REGION Network 63: BRAKE TEST FAULT AXIS 12
   RUNG wire#powerrail
      Contact( "DB1046_C22_BRAKE_TEST".BRAKE_TEST_ERROR )
      wire#w1
      Contact( #BRAKE_TEST_AXIS_C22 )
      wire#w2
      Coil( "DB1030_TEST_STOP".TEST_STP_TST_BRK_F_AX_12 )
   END_RUNG
   RUNG wire#powerrail
      Contact( "DB1030_TEST_STOP".TEST_STP_SQ_TIME_EXCEEDED )
      Contact( "DB1030_TEST_STOP".TEST_STP_TST_BRK_AX_12 )
   END_RUNG wire#w1
   RUNG wire#powerrail
      Contact( "DB1030_TEST_STOP".TEST_STP_TST_BRK_F_AX_12 )
      I_Contact( "DB2120_MPP_ITC_IPC".RESET_FAULTS )
   END_RUNG wire#w1
   RUNG wire#w2
      Coil( "DB426_ALARMS_WARNINGS".ALARMS.GENERAL."700603" )
   END_RUNG
   // the same network as SCL:
   "DB1030_TEST_STOP".TEST_STP_TST_BRK_F_AX_12 := ("DB1046_C22_BRAKE_TEST".BRAKE_TEST_ERROR OR ("DB1030_TEST_STOP".TEST_STP_SQ_TIME_EXCEEDED AND "DB1030_TEST_STOP".TEST_STP_TST_BRK_AX_12) OR ("DB1030_TEST_STOP".TEST_STP_TST_BRK_F_AX_12 AND NOT "DB2120_MPP_ITC_IPC".RESET_FAULTS)) AND #BRAKE_TEST_AXIS_C22;
   "DB426_ALARMS_WARNINGS".ALARMS.GENERAL."700603" := "DB1030_TEST_STOP".TEST_STP_TST_BRK_F_AX_12;
END_REGION

REGION Network 64: BRAKE TEST FAULT AXIS 13
   RUNG wire#powerrail
      Contact( "DB1047_C23_BRAKE_TEST".BRAKE_TEST_ERROR )
      wire#w1
      Contact( #BRAKE_TEST_AXIS_C23 )
      wire#w2
      Coil( "DB1030_TEST_STOP".TEST_STP_TST_BRK_F_AX_13 )
   END_RUNG
   RUNG wire#powerrail
      Contact( "DB1030_TEST_STOP".TEST_STP_SQ_TIME_EXCEEDED )
      Contact( "DB1030_TEST_STOP".TEST_STP_TST_BRK_AX_13 )
   END_RUNG wire#w1
   RUNG wire#powerrail
      Contact( "DB1030_TEST_STOP".TEST_STP_TST_BRK_F_AX_13 )
      I_Contact( "DB2120_MPP_ITC_IPC".RESET_FAULTS )
   END_RUNG wire#w1
   RUNG wire#w2
      Coil( "DB426_ALARMS_WARNINGS".ALARMS.GENERAL."700604" )
   END_RUNG
   // the same network as SCL:
   "DB1030_TEST_STOP".TEST_STP_TST_BRK_F_AX_13 := ("DB1047_C23_BRAKE_TEST".BRAKE_TEST_ERROR OR ("DB1030_TEST_STOP".TEST_STP_SQ_TIME_EXCEEDED AND "DB1030_TEST_STOP".TEST_STP_TST_BRK_AX_13) OR ("DB1030_TEST_STOP".TEST_STP_TST_BRK_F_AX_13 AND NOT "DB2120_MPP_ITC_IPC".RESET_FAULTS)) AND #BRAKE_TEST_AXIS_C23;
   "DB426_ALARMS_WARNINGS".ALARMS.GENERAL."700604" := "DB1030_TEST_STOP".TEST_STP_TST_BRK_F_AX_13;
END_REGION

REGION Network 65: BRAKE TEST FAULT AXIS 14
   RUNG wire#powerrail
      Contact( "DB1048_C24_BRAKE_TEST".BRAKE_TEST_ERROR )
      wire#w1
      Contact( #BRAKE_TEST_AXIS_C24 )
      wire#w2
      Coil( "DB1030_TEST_STOP".TEST_STP_TST_BRK_F_AX_14 )
   END_RUNG
   RUNG wire#powerrail
      Contact( "DB1030_TEST_STOP".TEST_STP_SQ_TIME_EXCEEDED )
      Contact( "DB1030_TEST_STOP".TEST_STP_TST_BRK_AX_14 )
   END_RUNG wire#w1
   RUNG wire#powerrail
      Contact( "DB1030_TEST_STOP".TEST_STP_TST_BRK_F_AX_14 )
      I_Contact( "DB2120_MPP_ITC_IPC".RESET_FAULTS )
   END_RUNG wire#w1
   RUNG wire#w2
      Coil( "DB426_ALARMS_WARNINGS".ALARMS.GENERAL."700605" )
   END_RUNG
   // the same network as SCL:
   "DB1030_TEST_STOP".TEST_STP_TST_BRK_F_AX_14 := ("DB1048_C24_BRAKE_TEST".BRAKE_TEST_ERROR OR ("DB1030_TEST_STOP".TEST_STP_SQ_TIME_EXCEEDED AND "DB1030_TEST_STOP".TEST_STP_TST_BRK_AX_14) OR ("DB1030_TEST_STOP".TEST_STP_TST_BRK_F_AX_14 AND NOT "DB2120_MPP_ITC_IPC".RESET_FAULTS)) AND #BRAKE_TEST_AXIS_C24;
   "DB426_ALARMS_WARNINGS".ALARMS.GENERAL."700605" := "DB1030_TEST_STOP".TEST_STP_TST_BRK_F_AX_14;
END_REGION

REGION Network 66: BRAKE TEST FAULT AXIS 15
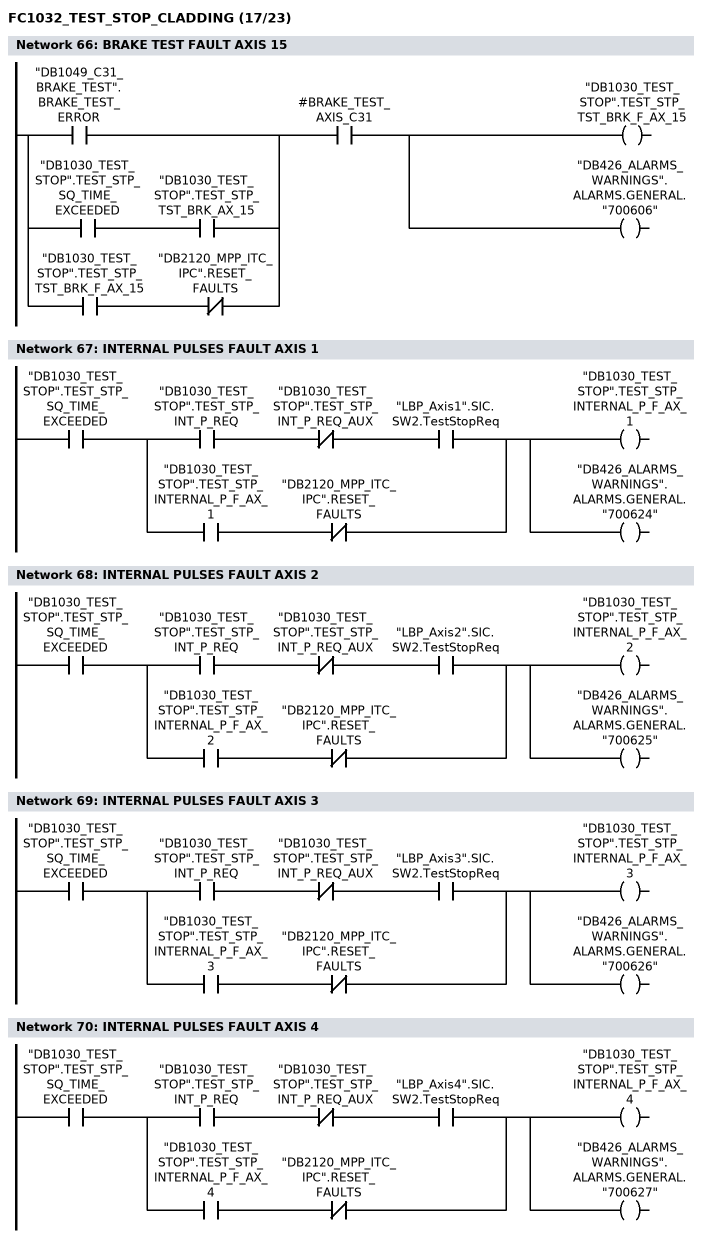
   RUNG wire#powerrail
      Contact( "DB1049_C31_BRAKE_TEST".BRAKE_TEST_ERROR )
      wire#w1
      Contact( #BRAKE_TEST_AXIS_C31 )
      wire#w2
      Coil( "DB1030_TEST_STOP".TEST_STP_TST_BRK_F_AX_15 )
   END_RUNG
   RUNG wire#powerrail
      Contact( "DB1030_TEST_STOP".TEST_STP_SQ_TIME_EXCEEDED )
      Contact( "DB1030_TEST_STOP".TEST_STP_TST_BRK_AX_15 )
   END_RUNG wire#w1
   RUNG wire#powerrail
      Contact( "DB1030_TEST_STOP".TEST_STP_TST_BRK_F_AX_15 )
      I_Contact( "DB2120_MPP_ITC_IPC".RESET_FAULTS )
   END_RUNG wire#w1
   RUNG wire#w2
      Coil( "DB426_ALARMS_WARNINGS".ALARMS.GENERAL."700606" )
   END_RUNG
   // the same network as SCL:
   "DB1030_TEST_STOP".TEST_STP_TST_BRK_F_AX_15 := ("DB1049_C31_BRAKE_TEST".BRAKE_TEST_ERROR OR ("DB1030_TEST_STOP".TEST_STP_SQ_TIME_EXCEEDED AND "DB1030_TEST_STOP".TEST_STP_TST_BRK_AX_15) OR ("DB1030_TEST_STOP".TEST_STP_TST_BRK_F_AX_15 AND NOT "DB2120_MPP_ITC_IPC".RESET_FAULTS)) AND #BRAKE_TEST_AXIS_C31;
   "DB426_ALARMS_WARNINGS".ALARMS.GENERAL."700606" := "DB1030_TEST_STOP".TEST_STP_TST_BRK_F_AX_15;
END_REGION

REGION Network 67: INTERNAL PULSES FAULT AXIS 1
   RUNG wire#powerrail
      Contact( "DB1030_TEST_STOP".TEST_STP_SQ_TIME_EXCEEDED )
      wire#w1
      Contact( "DB1030_TEST_STOP".TEST_STP_INT_P_REQ )
      I_Contact( "DB1030_TEST_STOP".TEST_STP_INT_P_REQ_AUX )
      Contact( "LBP_Axis1".SIC.SW2.TestStopReq )
      wire#w2
      Coil( "DB1030_TEST_STOP".TEST_STP_INTERNAL_P_F_AX_1 )
   END_RUNG
   RUNG wire#w1
      Contact( "DB1030_TEST_STOP".TEST_STP_INTERNAL_P_F_AX_1 )
      I_Contact( "DB2120_MPP_ITC_IPC".RESET_FAULTS )
   END_RUNG wire#w2
   RUNG wire#w2
      Coil( "DB426_ALARMS_WARNINGS".ALARMS.GENERAL."700624" )
   END_RUNG
   // the same network as SCL:
   "DB1030_TEST_STOP".TEST_STP_INTERNAL_P_F_AX_1 := "DB1030_TEST_STOP".TEST_STP_SQ_TIME_EXCEEDED AND (("DB1030_TEST_STOP".TEST_STP_INT_P_REQ AND NOT "DB1030_TEST_STOP".TEST_STP_INT_P_REQ_AUX AND "LBP_Axis1".SIC.SW2.TestStopReq) OR ("DB1030_TEST_STOP".TEST_STP_INTERNAL_P_F_AX_1 AND NOT "DB2120_MPP_ITC_IPC".RESET_FAULTS));
   "DB426_ALARMS_WARNINGS".ALARMS.GENERAL."700624" := "DB1030_TEST_STOP".TEST_STP_INTERNAL_P_F_AX_1;
END_REGION

REGION Network 68: INTERNAL PULSES FAULT AXIS 2
   RUNG wire#powerrail
      Contact( "DB1030_TEST_STOP".TEST_STP_SQ_TIME_EXCEEDED )
      wire#w1
      Contact( "DB1030_TEST_STOP".TEST_STP_INT_P_REQ )
      I_Contact( "DB1030_TEST_STOP".TEST_STP_INT_P_REQ_AUX )
      Contact( "LBP_Axis2".SIC.SW2.TestStopReq )
      wire#w2
      Coil( "DB1030_TEST_STOP".TEST_STP_INTERNAL_P_F_AX_2 )
   END_RUNG
   RUNG wire#w1
      Contact( "DB1030_TEST_STOP".TEST_STP_INTERNAL_P_F_AX_2 )
      I_Contact( "DB2120_MPP_ITC_IPC".RESET_FAULTS )
   END_RUNG wire#w2
   RUNG wire#w2
      Coil( "DB426_ALARMS_WARNINGS".ALARMS.GENERAL."700625" )
   END_RUNG
   // the same network as SCL:
   "DB1030_TEST_STOP".TEST_STP_INTERNAL_P_F_AX_2 := "DB1030_TEST_STOP".TEST_STP_SQ_TIME_EXCEEDED AND (("DB1030_TEST_STOP".TEST_STP_INT_P_REQ AND NOT "DB1030_TEST_STOP".TEST_STP_INT_P_REQ_AUX AND "LBP_Axis2".SIC.SW2.TestStopReq) OR ("DB1030_TEST_STOP".TEST_STP_INTERNAL_P_F_AX_2 AND NOT "DB2120_MPP_ITC_IPC".RESET_FAULTS));
   "DB426_ALARMS_WARNINGS".ALARMS.GENERAL."700625" := "DB1030_TEST_STOP".TEST_STP_INTERNAL_P_F_AX_2;
END_REGION

REGION Network 69: INTERNAL PULSES FAULT AXIS 3
   RUNG wire#powerrail
      Contact( "DB1030_TEST_STOP".TEST_STP_SQ_TIME_EXCEEDED )
      wire#w1
      Contact( "DB1030_TEST_STOP".TEST_STP_INT_P_REQ )
      I_Contact( "DB1030_TEST_STOP".TEST_STP_INT_P_REQ_AUX )
      Contact( "LBP_Axis3".SIC.SW2.TestStopReq )
      wire#w2
      Coil( "DB1030_TEST_STOP".TEST_STP_INTERNAL_P_F_AX_3 )
   END_RUNG
   RUNG wire#w1
      Contact( "DB1030_TEST_STOP".TEST_STP_INTERNAL_P_F_AX_3 )
      I_Contact( "DB2120_MPP_ITC_IPC".RESET_FAULTS )
   END_RUNG wire#w2
   RUNG wire#w2
      Coil( "DB426_ALARMS_WARNINGS".ALARMS.GENERAL."700626" )
   END_RUNG
   // the same network as SCL:
   "DB1030_TEST_STOP".TEST_STP_INTERNAL_P_F_AX_3 := "DB1030_TEST_STOP".TEST_STP_SQ_TIME_EXCEEDED AND (("DB1030_TEST_STOP".TEST_STP_INT_P_REQ AND NOT "DB1030_TEST_STOP".TEST_STP_INT_P_REQ_AUX AND "LBP_Axis3".SIC.SW2.TestStopReq) OR ("DB1030_TEST_STOP".TEST_STP_INTERNAL_P_F_AX_3 AND NOT "DB2120_MPP_ITC_IPC".RESET_FAULTS));
   "DB426_ALARMS_WARNINGS".ALARMS.GENERAL."700626" := "DB1030_TEST_STOP".TEST_STP_INTERNAL_P_F_AX_3;
END_REGION

REGION Network 70: INTERNAL PULSES FAULT AXIS 4
   RUNG wire#powerrail
      Contact( "DB1030_TEST_STOP".TEST_STP_SQ_TIME_EXCEEDED )
      wire#w1
      Contact( "DB1030_TEST_STOP".TEST_STP_INT_P_REQ )
      I_Contact( "DB1030_TEST_STOP".TEST_STP_INT_P_REQ_AUX )
      Contact( "LBP_Axis4".SIC.SW2.TestStopReq )
      wire#w2
      Coil( "DB1030_TEST_STOP".TEST_STP_INTERNAL_P_F_AX_4 )
   END_RUNG
   RUNG wire#w1
      Contact( "DB1030_TEST_STOP".TEST_STP_INTERNAL_P_F_AX_4 )
      I_Contact( "DB2120_MPP_ITC_IPC".RESET_FAULTS )
   END_RUNG wire#w2
   RUNG wire#w2
      Coil( "DB426_ALARMS_WARNINGS".ALARMS.GENERAL."700627" )
   END_RUNG
   // the same network as SCL:
   "DB1030_TEST_STOP".TEST_STP_INTERNAL_P_F_AX_4 := "DB1030_TEST_STOP".TEST_STP_SQ_TIME_EXCEEDED AND (("DB1030_TEST_STOP".TEST_STP_INT_P_REQ AND NOT "DB1030_TEST_STOP".TEST_STP_INT_P_REQ_AUX AND "LBP_Axis4".SIC.SW2.TestStopReq) OR ("DB1030_TEST_STOP".TEST_STP_INTERNAL_P_F_AX_4 AND NOT "DB2120_MPP_ITC_IPC".RESET_FAULTS));
   "DB426_ALARMS_WARNINGS".ALARMS.GENERAL."700627" := "DB1030_TEST_STOP".TEST_STP_INTERNAL_P_F_AX_4;
END_REGION

REGION Network 71: INTERNAL PULSES FAULT AXIS 5
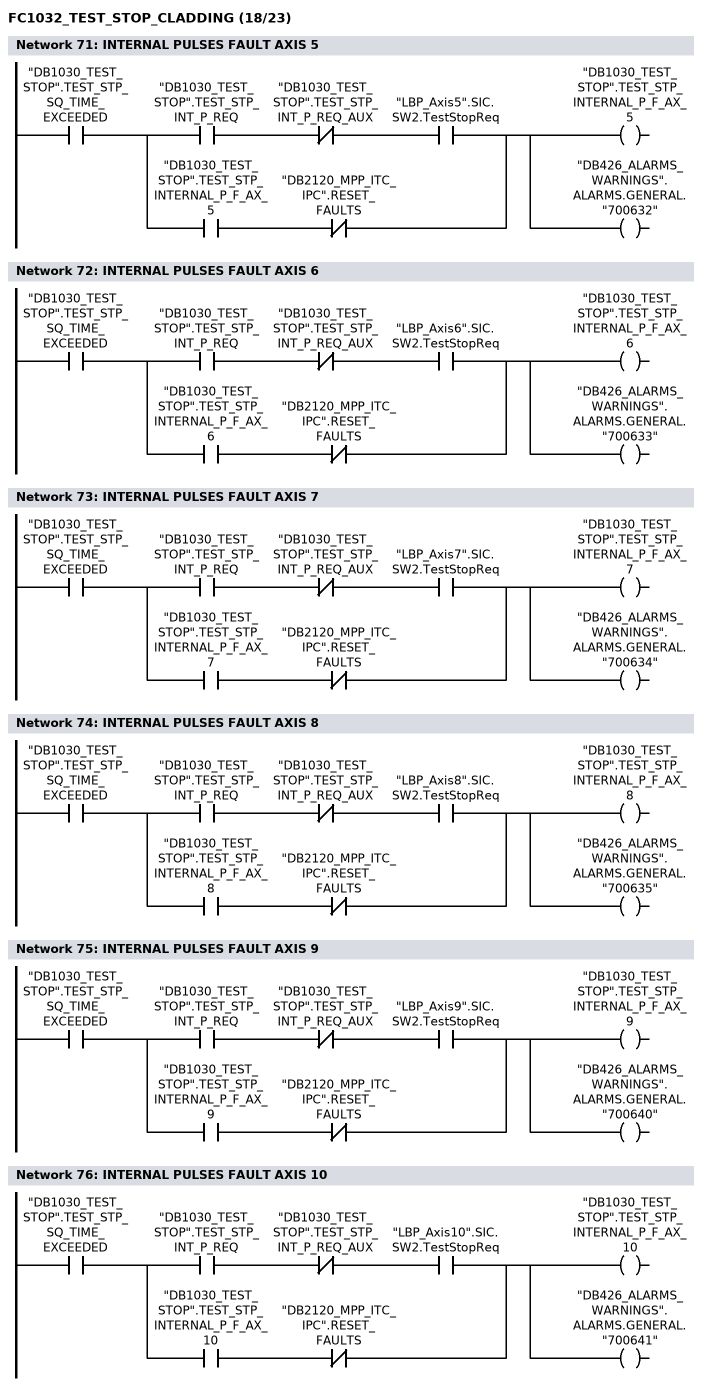
   RUNG wire#powerrail
      Contact( "DB1030_TEST_STOP".TEST_STP_SQ_TIME_EXCEEDED )
      wire#w1
      Contact( "DB1030_TEST_STOP".TEST_STP_INT_P_REQ )
      I_Contact( "DB1030_TEST_STOP".TEST_STP_INT_P_REQ_AUX )
      Contact( "LBP_Axis5".SIC.SW2.TestStopReq )
      wire#w2
      Coil( "DB1030_TEST_STOP".TEST_STP_INTERNAL_P_F_AX_5 )
   END_RUNG
   RUNG wire#w1
      Contact( "DB1030_TEST_STOP".TEST_STP_INTERNAL_P_F_AX_5 )
      I_Contact( "DB2120_MPP_ITC_IPC".RESET_FAULTS )
   END_RUNG wire#w2
   RUNG wire#w2
      Coil( "DB426_ALARMS_WARNINGS".ALARMS.GENERAL."700632" )
   END_RUNG
   // the same network as SCL:
   "DB1030_TEST_STOP".TEST_STP_INTERNAL_P_F_AX_5 := "DB1030_TEST_STOP".TEST_STP_SQ_TIME_EXCEEDED AND (("DB1030_TEST_STOP".TEST_STP_INT_P_REQ AND NOT "DB1030_TEST_STOP".TEST_STP_INT_P_REQ_AUX AND "LBP_Axis5".SIC.SW2.TestStopReq) OR ("DB1030_TEST_STOP".TEST_STP_INTERNAL_P_F_AX_5 AND NOT "DB2120_MPP_ITC_IPC".RESET_FAULTS));
   "DB426_ALARMS_WARNINGS".ALARMS.GENERAL."700632" := "DB1030_TEST_STOP".TEST_STP_INTERNAL_P_F_AX_5;
END_REGION

REGION Network 72: INTERNAL PULSES FAULT AXIS 6
   RUNG wire#powerrail
      Contact( "DB1030_TEST_STOP".TEST_STP_SQ_TIME_EXCEEDED )
      wire#w1
      Contact( "DB1030_TEST_STOP".TEST_STP_INT_P_REQ )
      I_Contact( "DB1030_TEST_STOP".TEST_STP_INT_P_REQ_AUX )
      Contact( "LBP_Axis6".SIC.SW2.TestStopReq )
      wire#w2
      Coil( "DB1030_TEST_STOP".TEST_STP_INTERNAL_P_F_AX_6 )
   END_RUNG
   RUNG wire#w1
      Contact( "DB1030_TEST_STOP".TEST_STP_INTERNAL_P_F_AX_6 )
      I_Contact( "DB2120_MPP_ITC_IPC".RESET_FAULTS )
   END_RUNG wire#w2
   RUNG wire#w2
      Coil( "DB426_ALARMS_WARNINGS".ALARMS.GENERAL."700633" )
   END_RUNG
   // the same network as SCL:
   "DB1030_TEST_STOP".TEST_STP_INTERNAL_P_F_AX_6 := "DB1030_TEST_STOP".TEST_STP_SQ_TIME_EXCEEDED AND (("DB1030_TEST_STOP".TEST_STP_INT_P_REQ AND NOT "DB1030_TEST_STOP".TEST_STP_INT_P_REQ_AUX AND "LBP_Axis6".SIC.SW2.TestStopReq) OR ("DB1030_TEST_STOP".TEST_STP_INTERNAL_P_F_AX_6 AND NOT "DB2120_MPP_ITC_IPC".RESET_FAULTS));
   "DB426_ALARMS_WARNINGS".ALARMS.GENERAL."700633" := "DB1030_TEST_STOP".TEST_STP_INTERNAL_P_F_AX_6;
END_REGION

REGION Network 73: INTERNAL PULSES FAULT AXIS 7
   RUNG wire#powerrail
      Contact( "DB1030_TEST_STOP".TEST_STP_SQ_TIME_EXCEEDED )
      wire#w1
      Contact( "DB1030_TEST_STOP".TEST_STP_INT_P_REQ )
      I_Contact( "DB1030_TEST_STOP".TEST_STP_INT_P_REQ_AUX )
      Contact( "LBP_Axis7".SIC.SW2.TestStopReq )
      wire#w2
      Coil( "DB1030_TEST_STOP".TEST_STP_INTERNAL_P_F_AX_7 )
   END_RUNG
   RUNG wire#w1
      Contact( "DB1030_TEST_STOP".TEST_STP_INTERNAL_P_F_AX_7 )
      I_Contact( "DB2120_MPP_ITC_IPC".RESET_FAULTS )
   END_RUNG wire#w2
   RUNG wire#w2
      Coil( "DB426_ALARMS_WARNINGS".ALARMS.GENERAL."700634" )
   END_RUNG
   // the same network as SCL:
   "DB1030_TEST_STOP".TEST_STP_INTERNAL_P_F_AX_7 := "DB1030_TEST_STOP".TEST_STP_SQ_TIME_EXCEEDED AND (("DB1030_TEST_STOP".TEST_STP_INT_P_REQ AND NOT "DB1030_TEST_STOP".TEST_STP_INT_P_REQ_AUX AND "LBP_Axis7".SIC.SW2.TestStopReq) OR ("DB1030_TEST_STOP".TEST_STP_INTERNAL_P_F_AX_7 AND NOT "DB2120_MPP_ITC_IPC".RESET_FAULTS));
   "DB426_ALARMS_WARNINGS".ALARMS.GENERAL."700634" := "DB1030_TEST_STOP".TEST_STP_INTERNAL_P_F_AX_7;
END_REGION

REGION Network 74: INTERNAL PULSES FAULT AXIS 8
   RUNG wire#powerrail
      Contact( "DB1030_TEST_STOP".TEST_STP_SQ_TIME_EXCEEDED )
      wire#w1
      Contact( "DB1030_TEST_STOP".TEST_STP_INT_P_REQ )
      I_Contact( "DB1030_TEST_STOP".TEST_STP_INT_P_REQ_AUX )
      Contact( "LBP_Axis8".SIC.SW2.TestStopReq )
      wire#w2
      Coil( "DB1030_TEST_STOP".TEST_STP_INTERNAL_P_F_AX_8 )
   END_RUNG
   RUNG wire#w1
      Contact( "DB1030_TEST_STOP".TEST_STP_INTERNAL_P_F_AX_8 )
      I_Contact( "DB2120_MPP_ITC_IPC".RESET_FAULTS )
   END_RUNG wire#w2
   RUNG wire#w2
      Coil( "DB426_ALARMS_WARNINGS".ALARMS.GENERAL."700635" )
   END_RUNG
   // the same network as SCL:
   "DB1030_TEST_STOP".TEST_STP_INTERNAL_P_F_AX_8 := "DB1030_TEST_STOP".TEST_STP_SQ_TIME_EXCEEDED AND (("DB1030_TEST_STOP".TEST_STP_INT_P_REQ AND NOT "DB1030_TEST_STOP".TEST_STP_INT_P_REQ_AUX AND "LBP_Axis8".SIC.SW2.TestStopReq) OR ("DB1030_TEST_STOP".TEST_STP_INTERNAL_P_F_AX_8 AND NOT "DB2120_MPP_ITC_IPC".RESET_FAULTS));
   "DB426_ALARMS_WARNINGS".ALARMS.GENERAL."700635" := "DB1030_TEST_STOP".TEST_STP_INTERNAL_P_F_AX_8;
END_REGION

REGION Network 75: INTERNAL PULSES FAULT AXIS 9
   RUNG wire#powerrail
      Contact( "DB1030_TEST_STOP".TEST_STP_SQ_TIME_EXCEEDED )
      wire#w1
      Contact( "DB1030_TEST_STOP".TEST_STP_INT_P_REQ )
      I_Contact( "DB1030_TEST_STOP".TEST_STP_INT_P_REQ_AUX )
      Contact( "LBP_Axis9".SIC.SW2.TestStopReq )
      wire#w2
      Coil( "DB1030_TEST_STOP".TEST_STP_INTERNAL_P_F_AX_9 )
   END_RUNG
   RUNG wire#w1
      Contact( "DB1030_TEST_STOP".TEST_STP_INTERNAL_P_F_AX_9 )
      I_Contact( "DB2120_MPP_ITC_IPC".RESET_FAULTS )
   END_RUNG wire#w2
   RUNG wire#w2
      Coil( "DB426_ALARMS_WARNINGS".ALARMS.GENERAL."700640" )
   END_RUNG
   // the same network as SCL:
   "DB1030_TEST_STOP".TEST_STP_INTERNAL_P_F_AX_9 := "DB1030_TEST_STOP".TEST_STP_SQ_TIME_EXCEEDED AND (("DB1030_TEST_STOP".TEST_STP_INT_P_REQ AND NOT "DB1030_TEST_STOP".TEST_STP_INT_P_REQ_AUX AND "LBP_Axis9".SIC.SW2.TestStopReq) OR ("DB1030_TEST_STOP".TEST_STP_INTERNAL_P_F_AX_9 AND NOT "DB2120_MPP_ITC_IPC".RESET_FAULTS));
   "DB426_ALARMS_WARNINGS".ALARMS.GENERAL."700640" := "DB1030_TEST_STOP".TEST_STP_INTERNAL_P_F_AX_9;
END_REGION

REGION Network 76: INTERNAL PULSES FAULT AXIS 10
   RUNG wire#powerrail
      Contact( "DB1030_TEST_STOP".TEST_STP_SQ_TIME_EXCEEDED )
      wire#w1
      Contact( "DB1030_TEST_STOP".TEST_STP_INT_P_REQ )
      I_Contact( "DB1030_TEST_STOP".TEST_STP_INT_P_REQ_AUX )
      Contact( "LBP_Axis10".SIC.SW2.TestStopReq )
      wire#w2
      Coil( "DB1030_TEST_STOP".TEST_STP_INTERNAL_P_F_AX_10 )
   END_RUNG
   RUNG wire#w1
      Contact( "DB1030_TEST_STOP".TEST_STP_INTERNAL_P_F_AX_10 )
      I_Contact( "DB2120_MPP_ITC_IPC".RESET_FAULTS )
   END_RUNG wire#w2
   RUNG wire#w2
      Coil( "DB426_ALARMS_WARNINGS".ALARMS.GENERAL."700641" )
   END_RUNG
   // the same network as SCL:
   "DB1030_TEST_STOP".TEST_STP_INTERNAL_P_F_AX_10 := "DB1030_TEST_STOP".TEST_STP_SQ_TIME_EXCEEDED AND (("DB1030_TEST_STOP".TEST_STP_INT_P_REQ AND NOT "DB1030_TEST_STOP".TEST_STP_INT_P_REQ_AUX AND "LBP_Axis10".SIC.SW2.TestStopReq) OR ("DB1030_TEST_STOP".TEST_STP_INTERNAL_P_F_AX_10 AND NOT "DB2120_MPP_ITC_IPC".RESET_FAULTS));
   "DB426_ALARMS_WARNINGS".ALARMS.GENERAL."700641" := "DB1030_TEST_STOP".TEST_STP_INTERNAL_P_F_AX_10;
END_REGION

REGION Network 77: INTERNAL PULSES FAULT AXIS 11
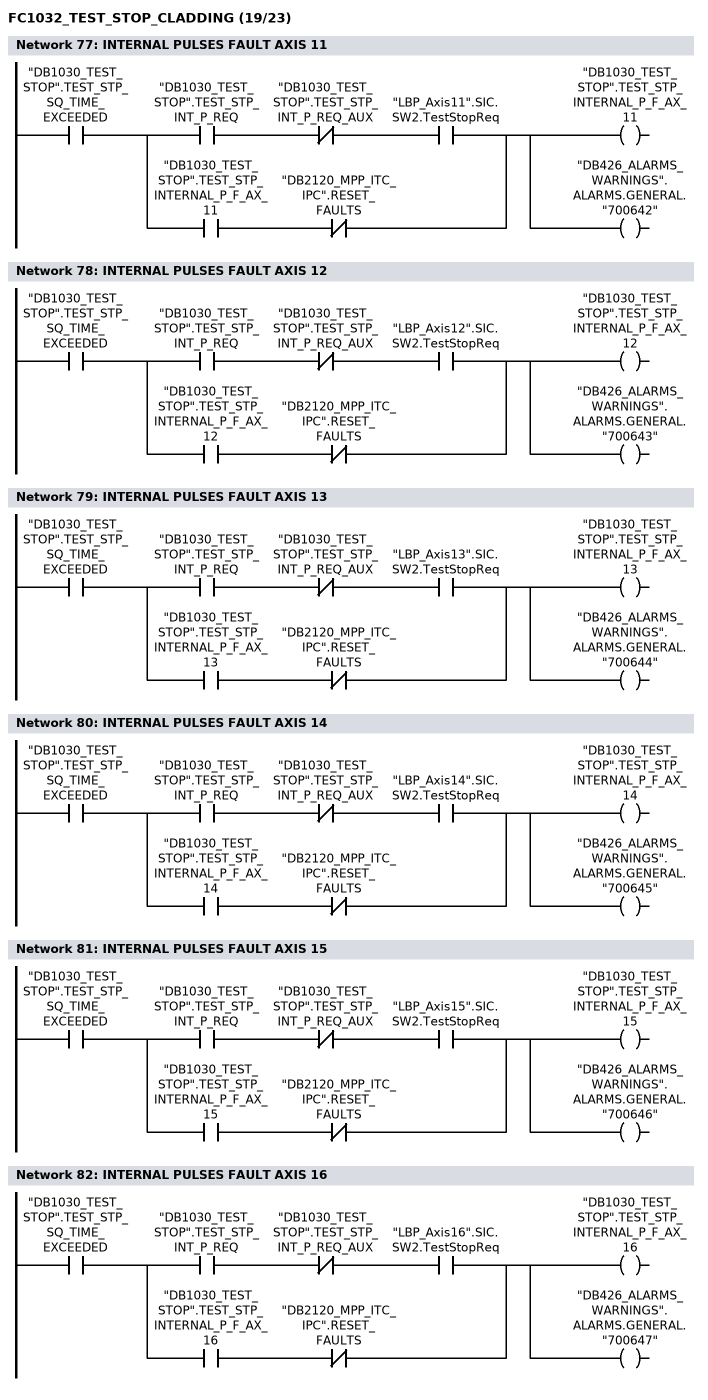
   RUNG wire#powerrail
      Contact( "DB1030_TEST_STOP".TEST_STP_SQ_TIME_EXCEEDED )
      wire#w1
      Contact( "DB1030_TEST_STOP".TEST_STP_INT_P_REQ )
      I_Contact( "DB1030_TEST_STOP".TEST_STP_INT_P_REQ_AUX )
      Contact( "LBP_Axis11".SIC.SW2.TestStopReq )
      wire#w2
      Coil( "DB1030_TEST_STOP".TEST_STP_INTERNAL_P_F_AX_11 )
   END_RUNG
   RUNG wire#w1
      Contact( "DB1030_TEST_STOP".TEST_STP_INTERNAL_P_F_AX_11 )
      I_Contact( "DB2120_MPP_ITC_IPC".RESET_FAULTS )
   END_RUNG wire#w2
   RUNG wire#w2
      Coil( "DB426_ALARMS_WARNINGS".ALARMS.GENERAL."700642" )
   END_RUNG
   // the same network as SCL:
   "DB1030_TEST_STOP".TEST_STP_INTERNAL_P_F_AX_11 := "DB1030_TEST_STOP".TEST_STP_SQ_TIME_EXCEEDED AND (("DB1030_TEST_STOP".TEST_STP_INT_P_REQ AND NOT "DB1030_TEST_STOP".TEST_STP_INT_P_REQ_AUX AND "LBP_Axis11".SIC.SW2.TestStopReq) OR ("DB1030_TEST_STOP".TEST_STP_INTERNAL_P_F_AX_11 AND NOT "DB2120_MPP_ITC_IPC".RESET_FAULTS));
   "DB426_ALARMS_WARNINGS".ALARMS.GENERAL."700642" := "DB1030_TEST_STOP".TEST_STP_INTERNAL_P_F_AX_11;
END_REGION

REGION Network 78: INTERNAL PULSES FAULT AXIS 12
   RUNG wire#powerrail
      Contact( "DB1030_TEST_STOP".TEST_STP_SQ_TIME_EXCEEDED )
      wire#w1
      Contact( "DB1030_TEST_STOP".TEST_STP_INT_P_REQ )
      I_Contact( "DB1030_TEST_STOP".TEST_STP_INT_P_REQ_AUX )
      Contact( "LBP_Axis12".SIC.SW2.TestStopReq )
      wire#w2
      Coil( "DB1030_TEST_STOP".TEST_STP_INTERNAL_P_F_AX_12 )
   END_RUNG
   RUNG wire#w1
      Contact( "DB1030_TEST_STOP".TEST_STP_INTERNAL_P_F_AX_12 )
      I_Contact( "DB2120_MPP_ITC_IPC".RESET_FAULTS )
   END_RUNG wire#w2
   RUNG wire#w2
      Coil( "DB426_ALARMS_WARNINGS".ALARMS.GENERAL."700643" )
   END_RUNG
   // the same network as SCL:
   "DB1030_TEST_STOP".TEST_STP_INTERNAL_P_F_AX_12 := "DB1030_TEST_STOP".TEST_STP_SQ_TIME_EXCEEDED AND (("DB1030_TEST_STOP".TEST_STP_INT_P_REQ AND NOT "DB1030_TEST_STOP".TEST_STP_INT_P_REQ_AUX AND "LBP_Axis12".SIC.SW2.TestStopReq) OR ("DB1030_TEST_STOP".TEST_STP_INTERNAL_P_F_AX_12 AND NOT "DB2120_MPP_ITC_IPC".RESET_FAULTS));
   "DB426_ALARMS_WARNINGS".ALARMS.GENERAL."700643" := "DB1030_TEST_STOP".TEST_STP_INTERNAL_P_F_AX_12;
END_REGION

REGION Network 79: INTERNAL PULSES FAULT AXIS 13
   RUNG wire#powerrail
      Contact( "DB1030_TEST_STOP".TEST_STP_SQ_TIME_EXCEEDED )
      wire#w1
      Contact( "DB1030_TEST_STOP".TEST_STP_INT_P_REQ )
      I_Contact( "DB1030_TEST_STOP".TEST_STP_INT_P_REQ_AUX )
      Contact( "LBP_Axis13".SIC.SW2.TestStopReq )
      wire#w2
      Coil( "DB1030_TEST_STOP".TEST_STP_INTERNAL_P_F_AX_13 )
   END_RUNG
   RUNG wire#w1
      Contact( "DB1030_TEST_STOP".TEST_STP_INTERNAL_P_F_AX_13 )
      I_Contact( "DB2120_MPP_ITC_IPC".RESET_FAULTS )
   END_RUNG wire#w2
   RUNG wire#w2
      Coil( "DB426_ALARMS_WARNINGS".ALARMS.GENERAL."700644" )
   END_RUNG
   // the same network as SCL:
   "DB1030_TEST_STOP".TEST_STP_INTERNAL_P_F_AX_13 := "DB1030_TEST_STOP".TEST_STP_SQ_TIME_EXCEEDED AND (("DB1030_TEST_STOP".TEST_STP_INT_P_REQ AND NOT "DB1030_TEST_STOP".TEST_STP_INT_P_REQ_AUX AND "LBP_Axis13".SIC.SW2.TestStopReq) OR ("DB1030_TEST_STOP".TEST_STP_INTERNAL_P_F_AX_13 AND NOT "DB2120_MPP_ITC_IPC".RESET_FAULTS));
   "DB426_ALARMS_WARNINGS".ALARMS.GENERAL."700644" := "DB1030_TEST_STOP".TEST_STP_INTERNAL_P_F_AX_13;
END_REGION

REGION Network 80: INTERNAL PULSES FAULT AXIS 14
   RUNG wire#powerrail
      Contact( "DB1030_TEST_STOP".TEST_STP_SQ_TIME_EXCEEDED )
      wire#w1
      Contact( "DB1030_TEST_STOP".TEST_STP_INT_P_REQ )
      I_Contact( "DB1030_TEST_STOP".TEST_STP_INT_P_REQ_AUX )
      Contact( "LBP_Axis14".SIC.SW2.TestStopReq )
      wire#w2
      Coil( "DB1030_TEST_STOP".TEST_STP_INTERNAL_P_F_AX_14 )
   END_RUNG
   RUNG wire#w1
      Contact( "DB1030_TEST_STOP".TEST_STP_INTERNAL_P_F_AX_14 )
      I_Contact( "DB2120_MPP_ITC_IPC".RESET_FAULTS )
   END_RUNG wire#w2
   RUNG wire#w2
      Coil( "DB426_ALARMS_WARNINGS".ALARMS.GENERAL."700645" )
   END_RUNG
   // the same network as SCL:
   "DB1030_TEST_STOP".TEST_STP_INTERNAL_P_F_AX_14 := "DB1030_TEST_STOP".TEST_STP_SQ_TIME_EXCEEDED AND (("DB1030_TEST_STOP".TEST_STP_INT_P_REQ AND NOT "DB1030_TEST_STOP".TEST_STP_INT_P_REQ_AUX AND "LBP_Axis14".SIC.SW2.TestStopReq) OR ("DB1030_TEST_STOP".TEST_STP_INTERNAL_P_F_AX_14 AND NOT "DB2120_MPP_ITC_IPC".RESET_FAULTS));
   "DB426_ALARMS_WARNINGS".ALARMS.GENERAL."700645" := "DB1030_TEST_STOP".TEST_STP_INTERNAL_P_F_AX_14;
END_REGION

REGION Network 81: INTERNAL PULSES FAULT AXIS 15
   RUNG wire#powerrail
      Contact( "DB1030_TEST_STOP".TEST_STP_SQ_TIME_EXCEEDED )
      wire#w1
      Contact( "DB1030_TEST_STOP".TEST_STP_INT_P_REQ )
      I_Contact( "DB1030_TEST_STOP".TEST_STP_INT_P_REQ_AUX )
      Contact( "LBP_Axis15".SIC.SW2.TestStopReq )
      wire#w2
      Coil( "DB1030_TEST_STOP".TEST_STP_INTERNAL_P_F_AX_15 )
   END_RUNG
   RUNG wire#w1
      Contact( "DB1030_TEST_STOP".TEST_STP_INTERNAL_P_F_AX_15 )
      I_Contact( "DB2120_MPP_ITC_IPC".RESET_FAULTS )
   END_RUNG wire#w2
   RUNG wire#w2
      Coil( "DB426_ALARMS_WARNINGS".ALARMS.GENERAL."700646" )
   END_RUNG
   // the same network as SCL:
   "DB1030_TEST_STOP".TEST_STP_INTERNAL_P_F_AX_15 := "DB1030_TEST_STOP".TEST_STP_SQ_TIME_EXCEEDED AND (("DB1030_TEST_STOP".TEST_STP_INT_P_REQ AND NOT "DB1030_TEST_STOP".TEST_STP_INT_P_REQ_AUX AND "LBP_Axis15".SIC.SW2.TestStopReq) OR ("DB1030_TEST_STOP".TEST_STP_INTERNAL_P_F_AX_15 AND NOT "DB2120_MPP_ITC_IPC".RESET_FAULTS));
   "DB426_ALARMS_WARNINGS".ALARMS.GENERAL."700646" := "DB1030_TEST_STOP".TEST_STP_INTERNAL_P_F_AX_15;
END_REGION

REGION Network 82: INTERNAL PULSES FAULT AXIS 16
   RUNG wire#powerrail
      Contact( "DB1030_TEST_STOP".TEST_STP_SQ_TIME_EXCEEDED )
      wire#w1
      Contact( "DB1030_TEST_STOP".TEST_STP_INT_P_REQ )
      I_Contact( "DB1030_TEST_STOP".TEST_STP_INT_P_REQ_AUX )
      Contact( "LBP_Axis16".SIC.SW2.TestStopReq )
      wire#w2
      Coil( "DB1030_TEST_STOP".TEST_STP_INTERNAL_P_F_AX_16 )
   END_RUNG
   RUNG wire#w1
      Contact( "DB1030_TEST_STOP".TEST_STP_INTERNAL_P_F_AX_16 )
      I_Contact( "DB2120_MPP_ITC_IPC".RESET_FAULTS )
   END_RUNG wire#w2
   RUNG wire#w2
      Coil( "DB426_ALARMS_WARNINGS".ALARMS.GENERAL."700647" )
   END_RUNG
   // the same network as SCL:
   "DB1030_TEST_STOP".TEST_STP_INTERNAL_P_F_AX_16 := "DB1030_TEST_STOP".TEST_STP_SQ_TIME_EXCEEDED AND (("DB1030_TEST_STOP".TEST_STP_INT_P_REQ AND NOT "DB1030_TEST_STOP".TEST_STP_INT_P_REQ_AUX AND "LBP_Axis16".SIC.SW2.TestStopReq) OR ("DB1030_TEST_STOP".TEST_STP_INTERNAL_P_F_AX_16 AND NOT "DB2120_MPP_ITC_IPC".RESET_FAULTS));
   "DB426_ALARMS_WARNINGS".ALARMS.GENERAL."700647" := "DB1030_TEST_STOP".TEST_STP_INTERNAL_P_F_AX_16;
END_REGION

REGION Network 83: INTERNAL PULSES FAULT AXIS 17
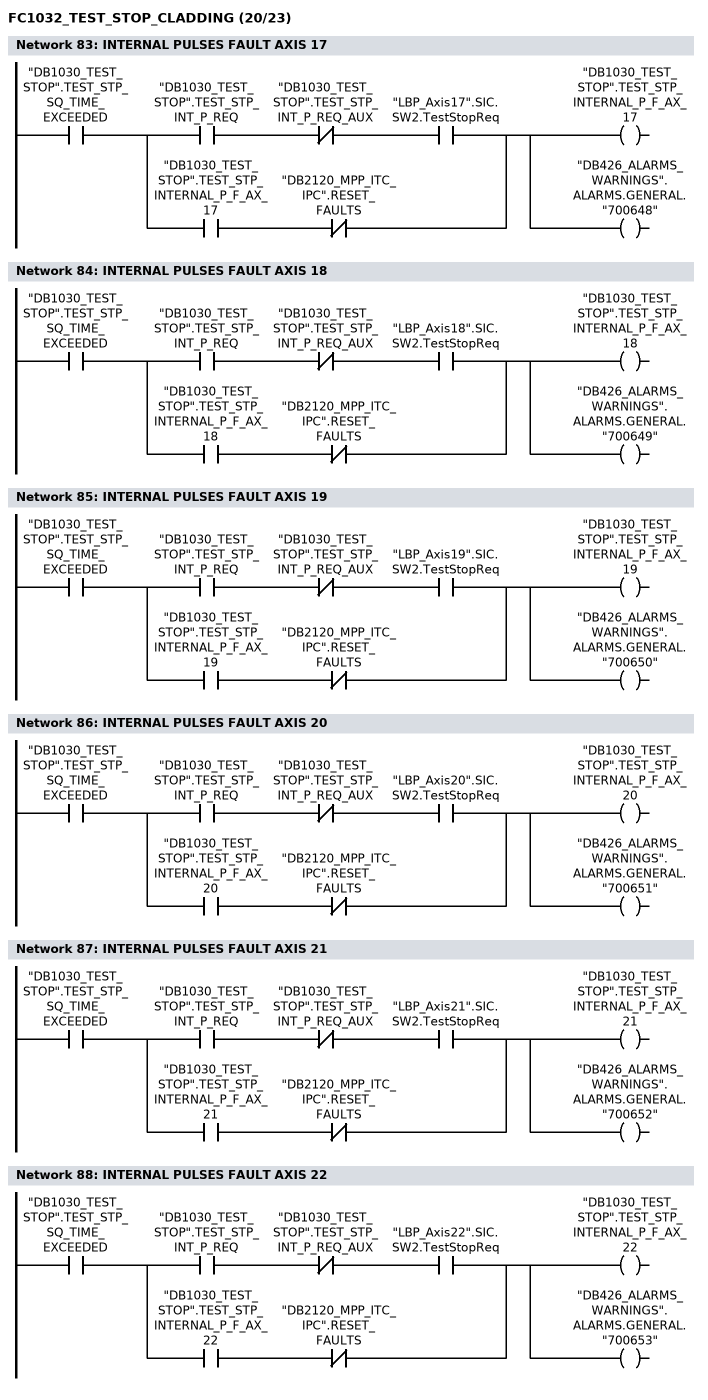
   RUNG wire#powerrail
      Contact( "DB1030_TEST_STOP".TEST_STP_SQ_TIME_EXCEEDED )
      wire#w1
      Contact( "DB1030_TEST_STOP".TEST_STP_INT_P_REQ )
      I_Contact( "DB1030_TEST_STOP".TEST_STP_INT_P_REQ_AUX )
      Contact( "LBP_Axis17".SIC.SW2.TestStopReq )
      wire#w2
      Coil( "DB1030_TEST_STOP".TEST_STP_INTERNAL_P_F_AX_17 )
   END_RUNG
   RUNG wire#w1
      Contact( "DB1030_TEST_STOP".TEST_STP_INTERNAL_P_F_AX_17 )
      I_Contact( "DB2120_MPP_ITC_IPC".RESET_FAULTS )
   END_RUNG wire#w2
   RUNG wire#w2
      Coil( "DB426_ALARMS_WARNINGS".ALARMS.GENERAL."700648" )
   END_RUNG
   // the same network as SCL:
   "DB1030_TEST_STOP".TEST_STP_INTERNAL_P_F_AX_17 := "DB1030_TEST_STOP".TEST_STP_SQ_TIME_EXCEEDED AND (("DB1030_TEST_STOP".TEST_STP_INT_P_REQ AND NOT "DB1030_TEST_STOP".TEST_STP_INT_P_REQ_AUX AND "LBP_Axis17".SIC.SW2.TestStopReq) OR ("DB1030_TEST_STOP".TEST_STP_INTERNAL_P_F_AX_17 AND NOT "DB2120_MPP_ITC_IPC".RESET_FAULTS));
   "DB426_ALARMS_WARNINGS".ALARMS.GENERAL."700648" := "DB1030_TEST_STOP".TEST_STP_INTERNAL_P_F_AX_17;
END_REGION

REGION Network 84: INTERNAL PULSES FAULT AXIS 18
   RUNG wire#powerrail
      Contact( "DB1030_TEST_STOP".TEST_STP_SQ_TIME_EXCEEDED )
      wire#w1
      Contact( "DB1030_TEST_STOP".TEST_STP_INT_P_REQ )
      I_Contact( "DB1030_TEST_STOP".TEST_STP_INT_P_REQ_AUX )
      Contact( "LBP_Axis18".SIC.SW2.TestStopReq )
      wire#w2
      Coil( "DB1030_TEST_STOP".TEST_STP_INTERNAL_P_F_AX_18 )
   END_RUNG
   RUNG wire#w1
      Contact( "DB1030_TEST_STOP".TEST_STP_INTERNAL_P_F_AX_18 )
      I_Contact( "DB2120_MPP_ITC_IPC".RESET_FAULTS )
   END_RUNG wire#w2
   RUNG wire#w2
      Coil( "DB426_ALARMS_WARNINGS".ALARMS.GENERAL."700649" )
   END_RUNG
   // the same network as SCL:
   "DB1030_TEST_STOP".TEST_STP_INTERNAL_P_F_AX_18 := "DB1030_TEST_STOP".TEST_STP_SQ_TIME_EXCEEDED AND (("DB1030_TEST_STOP".TEST_STP_INT_P_REQ AND NOT "DB1030_TEST_STOP".TEST_STP_INT_P_REQ_AUX AND "LBP_Axis18".SIC.SW2.TestStopReq) OR ("DB1030_TEST_STOP".TEST_STP_INTERNAL_P_F_AX_18 AND NOT "DB2120_MPP_ITC_IPC".RESET_FAULTS));
   "DB426_ALARMS_WARNINGS".ALARMS.GENERAL."700649" := "DB1030_TEST_STOP".TEST_STP_INTERNAL_P_F_AX_18;
END_REGION

REGION Network 85: INTERNAL PULSES FAULT AXIS 19
   RUNG wire#powerrail
      Contact( "DB1030_TEST_STOP".TEST_STP_SQ_TIME_EXCEEDED )
      wire#w1
      Contact( "DB1030_TEST_STOP".TEST_STP_INT_P_REQ )
      I_Contact( "DB1030_TEST_STOP".TEST_STP_INT_P_REQ_AUX )
      Contact( "LBP_Axis19".SIC.SW2.TestStopReq )
      wire#w2
      Coil( "DB1030_TEST_STOP".TEST_STP_INTERNAL_P_F_AX_19 )
   END_RUNG
   RUNG wire#w1
      Contact( "DB1030_TEST_STOP".TEST_STP_INTERNAL_P_F_AX_19 )
      I_Contact( "DB2120_MPP_ITC_IPC".RESET_FAULTS )
   END_RUNG wire#w2
   RUNG wire#w2
      Coil( "DB426_ALARMS_WARNINGS".ALARMS.GENERAL."700650" )
   END_RUNG
   // the same network as SCL:
   "DB1030_TEST_STOP".TEST_STP_INTERNAL_P_F_AX_19 := "DB1030_TEST_STOP".TEST_STP_SQ_TIME_EXCEEDED AND (("DB1030_TEST_STOP".TEST_STP_INT_P_REQ AND NOT "DB1030_TEST_STOP".TEST_STP_INT_P_REQ_AUX AND "LBP_Axis19".SIC.SW2.TestStopReq) OR ("DB1030_TEST_STOP".TEST_STP_INTERNAL_P_F_AX_19 AND NOT "DB2120_MPP_ITC_IPC".RESET_FAULTS));
   "DB426_ALARMS_WARNINGS".ALARMS.GENERAL."700650" := "DB1030_TEST_STOP".TEST_STP_INTERNAL_P_F_AX_19;
END_REGION

REGION Network 86: INTERNAL PULSES FAULT AXIS 20
   RUNG wire#powerrail
      Contact( "DB1030_TEST_STOP".TEST_STP_SQ_TIME_EXCEEDED )
      wire#w1
      Contact( "DB1030_TEST_STOP".TEST_STP_INT_P_REQ )
      I_Contact( "DB1030_TEST_STOP".TEST_STP_INT_P_REQ_AUX )
      Contact( "LBP_Axis20".SIC.SW2.TestStopReq )
      wire#w2
      Coil( "DB1030_TEST_STOP".TEST_STP_INTERNAL_P_F_AX_20 )
   END_RUNG
   RUNG wire#w1
      Contact( "DB1030_TEST_STOP".TEST_STP_INTERNAL_P_F_AX_20 )
      I_Contact( "DB2120_MPP_ITC_IPC".RESET_FAULTS )
   END_RUNG wire#w2
   RUNG wire#w2
      Coil( "DB426_ALARMS_WARNINGS".ALARMS.GENERAL."700651" )
   END_RUNG
   // the same network as SCL:
   "DB1030_TEST_STOP".TEST_STP_INTERNAL_P_F_AX_20 := "DB1030_TEST_STOP".TEST_STP_SQ_TIME_EXCEEDED AND (("DB1030_TEST_STOP".TEST_STP_INT_P_REQ AND NOT "DB1030_TEST_STOP".TEST_STP_INT_P_REQ_AUX AND "LBP_Axis20".SIC.SW2.TestStopReq) OR ("DB1030_TEST_STOP".TEST_STP_INTERNAL_P_F_AX_20 AND NOT "DB2120_MPP_ITC_IPC".RESET_FAULTS));
   "DB426_ALARMS_WARNINGS".ALARMS.GENERAL."700651" := "DB1030_TEST_STOP".TEST_STP_INTERNAL_P_F_AX_20;
END_REGION

REGION Network 87: INTERNAL PULSES FAULT AXIS 21
   RUNG wire#powerrail
      Contact( "DB1030_TEST_STOP".TEST_STP_SQ_TIME_EXCEEDED )
      wire#w1
      Contact( "DB1030_TEST_STOP".TEST_STP_INT_P_REQ )
      I_Contact( "DB1030_TEST_STOP".TEST_STP_INT_P_REQ_AUX )
      Contact( "LBP_Axis21".SIC.SW2.TestStopReq )
      wire#w2
      Coil( "DB1030_TEST_STOP".TEST_STP_INTERNAL_P_F_AX_21 )
   END_RUNG
   RUNG wire#w1
      Contact( "DB1030_TEST_STOP".TEST_STP_INTERNAL_P_F_AX_21 )
      I_Contact( "DB2120_MPP_ITC_IPC".RESET_FAULTS )
   END_RUNG wire#w2
   RUNG wire#w2
      Coil( "DB426_ALARMS_WARNINGS".ALARMS.GENERAL."700652" )
   END_RUNG
   // the same network as SCL:
   "DB1030_TEST_STOP".TEST_STP_INTERNAL_P_F_AX_21 := "DB1030_TEST_STOP".TEST_STP_SQ_TIME_EXCEEDED AND (("DB1030_TEST_STOP".TEST_STP_INT_P_REQ AND NOT "DB1030_TEST_STOP".TEST_STP_INT_P_REQ_AUX AND "LBP_Axis21".SIC.SW2.TestStopReq) OR ("DB1030_TEST_STOP".TEST_STP_INTERNAL_P_F_AX_21 AND NOT "DB2120_MPP_ITC_IPC".RESET_FAULTS));
   "DB426_ALARMS_WARNINGS".ALARMS.GENERAL."700652" := "DB1030_TEST_STOP".TEST_STP_INTERNAL_P_F_AX_21;
END_REGION

REGION Network 88: INTERNAL PULSES FAULT AXIS 22
   RUNG wire#powerrail
      Contact( "DB1030_TEST_STOP".TEST_STP_SQ_TIME_EXCEEDED )
      wire#w1
      Contact( "DB1030_TEST_STOP".TEST_STP_INT_P_REQ )
      I_Contact( "DB1030_TEST_STOP".TEST_STP_INT_P_REQ_AUX )
      Contact( "LBP_Axis22".SIC.SW2.TestStopReq )
      wire#w2
      Coil( "DB1030_TEST_STOP".TEST_STP_INTERNAL_P_F_AX_22 )
   END_RUNG
   RUNG wire#w1
      Contact( "DB1030_TEST_STOP".TEST_STP_INTERNAL_P_F_AX_22 )
      I_Contact( "DB2120_MPP_ITC_IPC".RESET_FAULTS )
   END_RUNG wire#w2
   RUNG wire#w2
      Coil( "DB426_ALARMS_WARNINGS".ALARMS.GENERAL."700653" )
   END_RUNG
   // the same network as SCL:
   "DB1030_TEST_STOP".TEST_STP_INTERNAL_P_F_AX_22 := "DB1030_TEST_STOP".TEST_STP_SQ_TIME_EXCEEDED AND (("DB1030_TEST_STOP".TEST_STP_INT_P_REQ AND NOT "DB1030_TEST_STOP".TEST_STP_INT_P_REQ_AUX AND "LBP_Axis22".SIC.SW2.TestStopReq) OR ("DB1030_TEST_STOP".TEST_STP_INTERNAL_P_F_AX_22 AND NOT "DB2120_MPP_ITC_IPC".RESET_FAULTS));
   "DB426_ALARMS_WARNINGS".ALARMS.GENERAL."700653" := "DB1030_TEST_STOP".TEST_STP_INTERNAL_P_F_AX_22;
END_REGION

REGION Network 89: INTERNAL PULSES FAULT AXIS 23
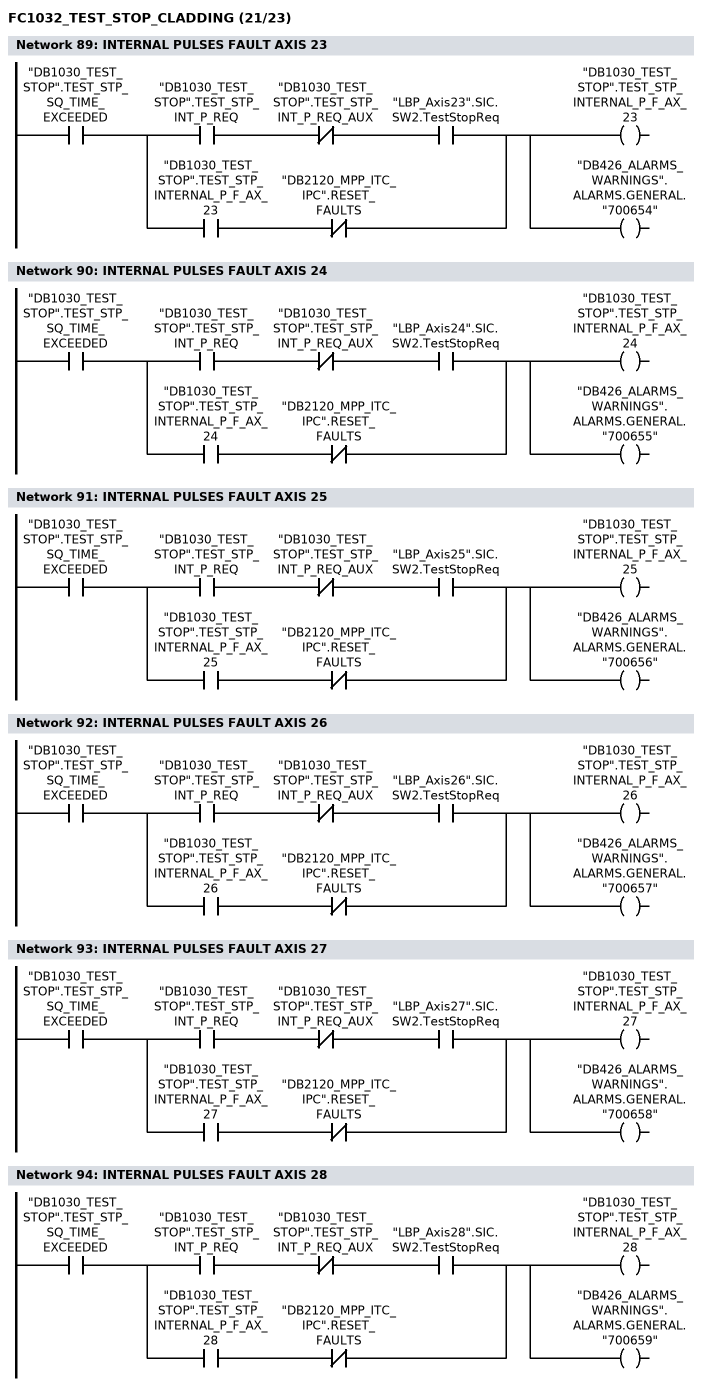
   RUNG wire#powerrail
      Contact( "DB1030_TEST_STOP".TEST_STP_SQ_TIME_EXCEEDED )
      wire#w1
      Contact( "DB1030_TEST_STOP".TEST_STP_INT_P_REQ )
      I_Contact( "DB1030_TEST_STOP".TEST_STP_INT_P_REQ_AUX )
      Contact( "LBP_Axis23".SIC.SW2.TestStopReq )
      wire#w2
      Coil( "DB1030_TEST_STOP".TEST_STP_INTERNAL_P_F_AX_23 )
   END_RUNG
   RUNG wire#w1
      Contact( "DB1030_TEST_STOP".TEST_STP_INTERNAL_P_F_AX_23 )
      I_Contact( "DB2120_MPP_ITC_IPC".RESET_FAULTS )
   END_RUNG wire#w2
   RUNG wire#w2
      Coil( "DB426_ALARMS_WARNINGS".ALARMS.GENERAL."700654" )
   END_RUNG
   // the same network as SCL:
   "DB1030_TEST_STOP".TEST_STP_INTERNAL_P_F_AX_23 := "DB1030_TEST_STOP".TEST_STP_SQ_TIME_EXCEEDED AND (("DB1030_TEST_STOP".TEST_STP_INT_P_REQ AND NOT "DB1030_TEST_STOP".TEST_STP_INT_P_REQ_AUX AND "LBP_Axis23".SIC.SW2.TestStopReq) OR ("DB1030_TEST_STOP".TEST_STP_INTERNAL_P_F_AX_23 AND NOT "DB2120_MPP_ITC_IPC".RESET_FAULTS));
   "DB426_ALARMS_WARNINGS".ALARMS.GENERAL."700654" := "DB1030_TEST_STOP".TEST_STP_INTERNAL_P_F_AX_23;
END_REGION

REGION Network 90: INTERNAL PULSES FAULT AXIS 24
   RUNG wire#powerrail
      Contact( "DB1030_TEST_STOP".TEST_STP_SQ_TIME_EXCEEDED )
      wire#w1
      Contact( "DB1030_TEST_STOP".TEST_STP_INT_P_REQ )
      I_Contact( "DB1030_TEST_STOP".TEST_STP_INT_P_REQ_AUX )
      Contact( "LBP_Axis24".SIC.SW2.TestStopReq )
      wire#w2
      Coil( "DB1030_TEST_STOP".TEST_STP_INTERNAL_P_F_AX_24 )
   END_RUNG
   RUNG wire#w1
      Contact( "DB1030_TEST_STOP".TEST_STP_INTERNAL_P_F_AX_24 )
      I_Contact( "DB2120_MPP_ITC_IPC".RESET_FAULTS )
   END_RUNG wire#w2
   RUNG wire#w2
      Coil( "DB426_ALARMS_WARNINGS".ALARMS.GENERAL."700655" )
   END_RUNG
   // the same network as SCL:
   "DB1030_TEST_STOP".TEST_STP_INTERNAL_P_F_AX_24 := "DB1030_TEST_STOP".TEST_STP_SQ_TIME_EXCEEDED AND (("DB1030_TEST_STOP".TEST_STP_INT_P_REQ AND NOT "DB1030_TEST_STOP".TEST_STP_INT_P_REQ_AUX AND "LBP_Axis24".SIC.SW2.TestStopReq) OR ("DB1030_TEST_STOP".TEST_STP_INTERNAL_P_F_AX_24 AND NOT "DB2120_MPP_ITC_IPC".RESET_FAULTS));
   "DB426_ALARMS_WARNINGS".ALARMS.GENERAL."700655" := "DB1030_TEST_STOP".TEST_STP_INTERNAL_P_F_AX_24;
END_REGION

REGION Network 91: INTERNAL PULSES FAULT AXIS 25
   RUNG wire#powerrail
      Contact( "DB1030_TEST_STOP".TEST_STP_SQ_TIME_EXCEEDED )
      wire#w1
      Contact( "DB1030_TEST_STOP".TEST_STP_INT_P_REQ )
      I_Contact( "DB1030_TEST_STOP".TEST_STP_INT_P_REQ_AUX )
      Contact( "LBP_Axis25".SIC.SW2.TestStopReq )
      wire#w2
      Coil( "DB1030_TEST_STOP".TEST_STP_INTERNAL_P_F_AX_25 )
   END_RUNG
   RUNG wire#w1
      Contact( "DB1030_TEST_STOP".TEST_STP_INTERNAL_P_F_AX_25 )
      I_Contact( "DB2120_MPP_ITC_IPC".RESET_FAULTS )
   END_RUNG wire#w2
   RUNG wire#w2
      Coil( "DB426_ALARMS_WARNINGS".ALARMS.GENERAL."700656" )
   END_RUNG
   // the same network as SCL:
   "DB1030_TEST_STOP".TEST_STP_INTERNAL_P_F_AX_25 := "DB1030_TEST_STOP".TEST_STP_SQ_TIME_EXCEEDED AND (("DB1030_TEST_STOP".TEST_STP_INT_P_REQ AND NOT "DB1030_TEST_STOP".TEST_STP_INT_P_REQ_AUX AND "LBP_Axis25".SIC.SW2.TestStopReq) OR ("DB1030_TEST_STOP".TEST_STP_INTERNAL_P_F_AX_25 AND NOT "DB2120_MPP_ITC_IPC".RESET_FAULTS));
   "DB426_ALARMS_WARNINGS".ALARMS.GENERAL."700656" := "DB1030_TEST_STOP".TEST_STP_INTERNAL_P_F_AX_25;
END_REGION

REGION Network 92: INTERNAL PULSES FAULT AXIS 26
   RUNG wire#powerrail
      Contact( "DB1030_TEST_STOP".TEST_STP_SQ_TIME_EXCEEDED )
      wire#w1
      Contact( "DB1030_TEST_STOP".TEST_STP_INT_P_REQ )
      I_Contact( "DB1030_TEST_STOP".TEST_STP_INT_P_REQ_AUX )
      Contact( "LBP_Axis26".SIC.SW2.TestStopReq )
      wire#w2
      Coil( "DB1030_TEST_STOP".TEST_STP_INTERNAL_P_F_AX_26 )
   END_RUNG
   RUNG wire#w1
      Contact( "DB1030_TEST_STOP".TEST_STP_INTERNAL_P_F_AX_26 )
      I_Contact( "DB2120_MPP_ITC_IPC".RESET_FAULTS )
   END_RUNG wire#w2
   RUNG wire#w2
      Coil( "DB426_ALARMS_WARNINGS".ALARMS.GENERAL."700657" )
   END_RUNG
   // the same network as SCL:
   "DB1030_TEST_STOP".TEST_STP_INTERNAL_P_F_AX_26 := "DB1030_TEST_STOP".TEST_STP_SQ_TIME_EXCEEDED AND (("DB1030_TEST_STOP".TEST_STP_INT_P_REQ AND NOT "DB1030_TEST_STOP".TEST_STP_INT_P_REQ_AUX AND "LBP_Axis26".SIC.SW2.TestStopReq) OR ("DB1030_TEST_STOP".TEST_STP_INTERNAL_P_F_AX_26 AND NOT "DB2120_MPP_ITC_IPC".RESET_FAULTS));
   "DB426_ALARMS_WARNINGS".ALARMS.GENERAL."700657" := "DB1030_TEST_STOP".TEST_STP_INTERNAL_P_F_AX_26;
END_REGION

REGION Network 93: INTERNAL PULSES FAULT AXIS 27
   RUNG wire#powerrail
      Contact( "DB1030_TEST_STOP".TEST_STP_SQ_TIME_EXCEEDED )
      wire#w1
      Contact( "DB1030_TEST_STOP".TEST_STP_INT_P_REQ )
      I_Contact( "DB1030_TEST_STOP".TEST_STP_INT_P_REQ_AUX )
      Contact( "LBP_Axis27".SIC.SW2.TestStopReq )
      wire#w2
      Coil( "DB1030_TEST_STOP".TEST_STP_INTERNAL_P_F_AX_27 )
   END_RUNG
   RUNG wire#w1
      Contact( "DB1030_TEST_STOP".TEST_STP_INTERNAL_P_F_AX_27 )
      I_Contact( "DB2120_MPP_ITC_IPC".RESET_FAULTS )
   END_RUNG wire#w2
   RUNG wire#w2
      Coil( "DB426_ALARMS_WARNINGS".ALARMS.GENERAL."700658" )
   END_RUNG
   // the same network as SCL:
   "DB1030_TEST_STOP".TEST_STP_INTERNAL_P_F_AX_27 := "DB1030_TEST_STOP".TEST_STP_SQ_TIME_EXCEEDED AND (("DB1030_TEST_STOP".TEST_STP_INT_P_REQ AND NOT "DB1030_TEST_STOP".TEST_STP_INT_P_REQ_AUX AND "LBP_Axis27".SIC.SW2.TestStopReq) OR ("DB1030_TEST_STOP".TEST_STP_INTERNAL_P_F_AX_27 AND NOT "DB2120_MPP_ITC_IPC".RESET_FAULTS));
   "DB426_ALARMS_WARNINGS".ALARMS.GENERAL."700658" := "DB1030_TEST_STOP".TEST_STP_INTERNAL_P_F_AX_27;
END_REGION

REGION Network 94: INTERNAL PULSES FAULT AXIS 28
   RUNG wire#powerrail
      Contact( "DB1030_TEST_STOP".TEST_STP_SQ_TIME_EXCEEDED )
      wire#w1
      Contact( "DB1030_TEST_STOP".TEST_STP_INT_P_REQ )
      I_Contact( "DB1030_TEST_STOP".TEST_STP_INT_P_REQ_AUX )
      Contact( "LBP_Axis28".SIC.SW2.TestStopReq )
      wire#w2
      Coil( "DB1030_TEST_STOP".TEST_STP_INTERNAL_P_F_AX_28 )
   END_RUNG
   RUNG wire#w1
      Contact( "DB1030_TEST_STOP".TEST_STP_INTERNAL_P_F_AX_28 )
      I_Contact( "DB2120_MPP_ITC_IPC".RESET_FAULTS )
   END_RUNG wire#w2
   RUNG wire#w2
      Coil( "DB426_ALARMS_WARNINGS".ALARMS.GENERAL."700659" )
   END_RUNG
   // the same network as SCL:
   "DB1030_TEST_STOP".TEST_STP_INTERNAL_P_F_AX_28 := "DB1030_TEST_STOP".TEST_STP_SQ_TIME_EXCEEDED AND (("DB1030_TEST_STOP".TEST_STP_INT_P_REQ AND NOT "DB1030_TEST_STOP".TEST_STP_INT_P_REQ_AUX AND "LBP_Axis28".SIC.SW2.TestStopReq) OR ("DB1030_TEST_STOP".TEST_STP_INTERNAL_P_F_AX_28 AND NOT "DB2120_MPP_ITC_IPC".RESET_FAULTS));
   "DB426_ALARMS_WARNINGS".ALARMS.GENERAL."700659" := "DB1030_TEST_STOP".TEST_STP_INTERNAL_P_F_AX_28;
END_REGION

REGION Network 95: INTERNAL PULSES FAULT AXIS 29
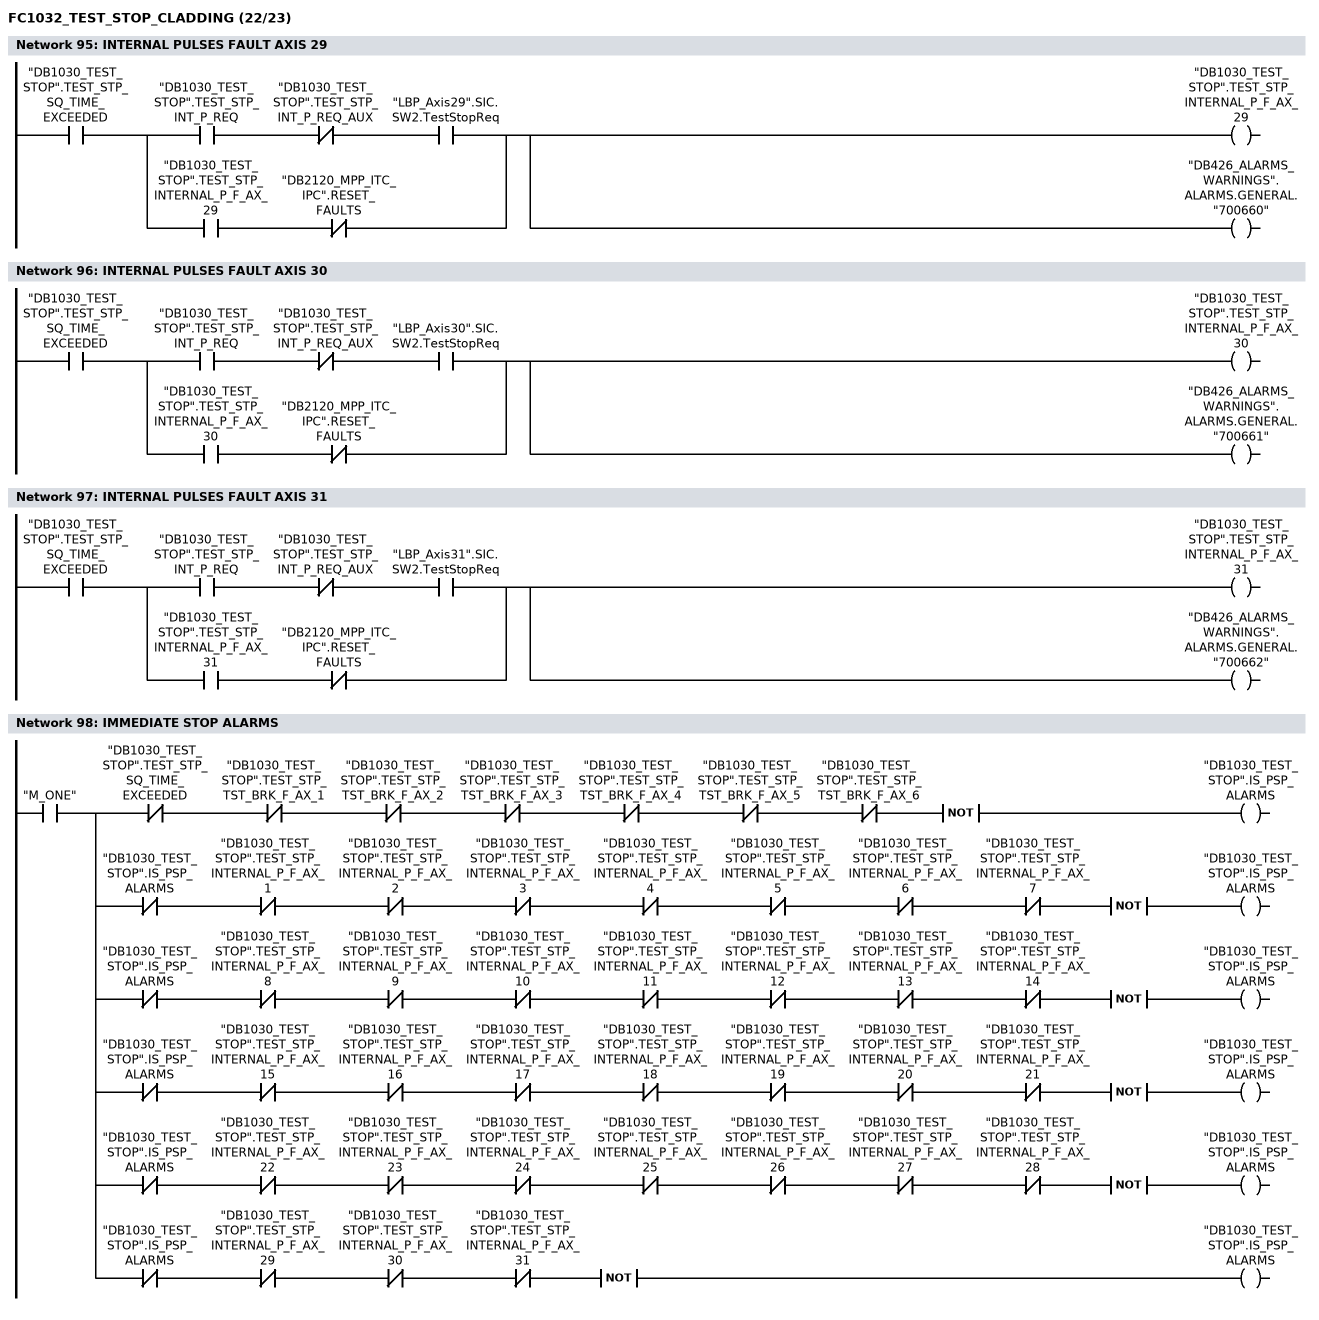
   RUNG wire#powerrail
      Contact( "DB1030_TEST_STOP".TEST_STP_SQ_TIME_EXCEEDED )
      wire#w1
      Contact( "DB1030_TEST_STOP".TEST_STP_INT_P_REQ )
      I_Contact( "DB1030_TEST_STOP".TEST_STP_INT_P_REQ_AUX )
      Contact( "LBP_Axis29".SIC.SW2.TestStopReq )
      wire#w2
      Coil( "DB1030_TEST_STOP".TEST_STP_INTERNAL_P_F_AX_29 )
   END_RUNG
   RUNG wire#w1
      Contact( "DB1030_TEST_STOP".TEST_STP_INTERNAL_P_F_AX_29 )
      I_Contact( "DB2120_MPP_ITC_IPC".RESET_FAULTS )
   END_RUNG wire#w2
   RUNG wire#w2
      Coil( "DB426_ALARMS_WARNINGS".ALARMS.GENERAL."700660" )
   END_RUNG
   // the same network as SCL:
   "DB1030_TEST_STOP".TEST_STP_INTERNAL_P_F_AX_29 := "DB1030_TEST_STOP".TEST_STP_SQ_TIME_EXCEEDED AND (("DB1030_TEST_STOP".TEST_STP_INT_P_REQ AND NOT "DB1030_TEST_STOP".TEST_STP_INT_P_REQ_AUX AND "LBP_Axis29".SIC.SW2.TestStopReq) OR ("DB1030_TEST_STOP".TEST_STP_INTERNAL_P_F_AX_29 AND NOT "DB2120_MPP_ITC_IPC".RESET_FAULTS));
   "DB426_ALARMS_WARNINGS".ALARMS.GENERAL."700660" := "DB1030_TEST_STOP".TEST_STP_INTERNAL_P_F_AX_29;
END_REGION

REGION Network 96: INTERNAL PULSES FAULT AXIS 30
   RUNG wire#powerrail
      Contact( "DB1030_TEST_STOP".TEST_STP_SQ_TIME_EXCEEDED )
      wire#w1
      Contact( "DB1030_TEST_STOP".TEST_STP_INT_P_REQ )
      I_Contact( "DB1030_TEST_STOP".TEST_STP_INT_P_REQ_AUX )
      Contact( "LBP_Axis30".SIC.SW2.TestStopReq )
      wire#w2
      Coil( "DB1030_TEST_STOP".TEST_STP_INTERNAL_P_F_AX_30 )
   END_RUNG
   RUNG wire#w1
      Contact( "DB1030_TEST_STOP".TEST_STP_INTERNAL_P_F_AX_30 )
      I_Contact( "DB2120_MPP_ITC_IPC".RESET_FAULTS )
   END_RUNG wire#w2
   RUNG wire#w2
      Coil( "DB426_ALARMS_WARNINGS".ALARMS.GENERAL."700661" )
   END_RUNG
   // the same network as SCL:
   "DB1030_TEST_STOP".TEST_STP_INTERNAL_P_F_AX_30 := "DB1030_TEST_STOP".TEST_STP_SQ_TIME_EXCEEDED AND (("DB1030_TEST_STOP".TEST_STP_INT_P_REQ AND NOT "DB1030_TEST_STOP".TEST_STP_INT_P_REQ_AUX AND "LBP_Axis30".SIC.SW2.TestStopReq) OR ("DB1030_TEST_STOP".TEST_STP_INTERNAL_P_F_AX_30 AND NOT "DB2120_MPP_ITC_IPC".RESET_FAULTS));
   "DB426_ALARMS_WARNINGS".ALARMS.GENERAL."700661" := "DB1030_TEST_STOP".TEST_STP_INTERNAL_P_F_AX_30;
END_REGION

REGION Network 97: INTERNAL PULSES FAULT AXIS 31
   RUNG wire#powerrail
      Contact( "DB1030_TEST_STOP".TEST_STP_SQ_TIME_EXCEEDED )
      wire#w1
      Contact( "DB1030_TEST_STOP".TEST_STP_INT_P_REQ )
      I_Contact( "DB1030_TEST_STOP".TEST_STP_INT_P_REQ_AUX )
      Contact( "LBP_Axis31".SIC.SW2.TestStopReq )
      wire#w2
      Coil( "DB1030_TEST_STOP".TEST_STP_INTERNAL_P_F_AX_31 )
   END_RUNG
   RUNG wire#w1
      Contact( "DB1030_TEST_STOP".TEST_STP_INTERNAL_P_F_AX_31 )
      I_Contact( "DB2120_MPP_ITC_IPC".RESET_FAULTS )
   END_RUNG wire#w2
   RUNG wire#w2
      Coil( "DB426_ALARMS_WARNINGS".ALARMS.GENERAL."700662" )
   END_RUNG
   // the same network as SCL:
   "DB1030_TEST_STOP".TEST_STP_INTERNAL_P_F_AX_31 := "DB1030_TEST_STOP".TEST_STP_SQ_TIME_EXCEEDED AND (("DB1030_TEST_STOP".TEST_STP_INT_P_REQ AND NOT "DB1030_TEST_STOP".TEST_STP_INT_P_REQ_AUX AND "LBP_Axis31".SIC.SW2.TestStopReq) OR ("DB1030_TEST_STOP".TEST_STP_INTERNAL_P_F_AX_31 AND NOT "DB2120_MPP_ITC_IPC".RESET_FAULTS));
   "DB426_ALARMS_WARNINGS".ALARMS.GENERAL."700662" := "DB1030_TEST_STOP".TEST_STP_INTERNAL_P_F_AX_31;
END_REGION

REGION Network 98: IMMEDIATE STOP ALARMS
   RUNG wire#powerrail
      Contact( "M_ONE" )
      wire#w1
      I_Contact( "DB1030_TEST_STOP".TEST_STP_SQ_TIME_EXCEEDED )
      I_Contact( "DB1030_TEST_STOP".TEST_STP_TST_BRK_F_AX_1 )
      I_Contact( "DB1030_TEST_STOP".TEST_STP_TST_BRK_F_AX_2 )
      I_Contact( "DB1030_TEST_STOP".TEST_STP_TST_BRK_F_AX_3 )
      I_Contact( "DB1030_TEST_STOP".TEST_STP_TST_BRK_F_AX_4 )
      I_Contact( "DB1030_TEST_STOP".TEST_STP_TST_BRK_F_AX_5 )
      I_Contact( "DB1030_TEST_STOP".TEST_STP_TST_BRK_F_AX_6 )
      Not()
      Coil( "DB1030_TEST_STOP".IS_PSP_ALARMS )
   END_RUNG
   RUNG wire#w1
      I_Contact( "DB1030_TEST_STOP".IS_PSP_ALARMS )
      I_Contact( "DB1030_TEST_STOP".TEST_STP_INTERNAL_P_F_AX_1 )
      I_Contact( "DB1030_TEST_STOP".TEST_STP_INTERNAL_P_F_AX_2 )
      I_Contact( "DB1030_TEST_STOP".TEST_STP_INTERNAL_P_F_AX_3 )
      I_Contact( "DB1030_TEST_STOP".TEST_STP_INTERNAL_P_F_AX_4 )
      I_Contact( "DB1030_TEST_STOP".TEST_STP_INTERNAL_P_F_AX_5 )
      I_Contact( "DB1030_TEST_STOP".TEST_STP_INTERNAL_P_F_AX_6 )
      I_Contact( "DB1030_TEST_STOP".TEST_STP_INTERNAL_P_F_AX_7 )
      Not()
      Coil( "DB1030_TEST_STOP".IS_PSP_ALARMS )
   END_RUNG
   RUNG wire#w1
      I_Contact( "DB1030_TEST_STOP".IS_PSP_ALARMS )
      I_Contact( "DB1030_TEST_STOP".TEST_STP_INTERNAL_P_F_AX_8 )
      I_Contact( "DB1030_TEST_STOP".TEST_STP_INTERNAL_P_F_AX_9 )
      I_Contact( "DB1030_TEST_STOP".TEST_STP_INTERNAL_P_F_AX_10 )
      I_Contact( "DB1030_TEST_STOP".TEST_STP_INTERNAL_P_F_AX_11 )
      I_Contact( "DB1030_TEST_STOP".TEST_STP_INTERNAL_P_F_AX_12 )
      I_Contact( "DB1030_TEST_STOP".TEST_STP_INTERNAL_P_F_AX_13 )
      I_Contact( "DB1030_TEST_STOP".TEST_STP_INTERNAL_P_F_AX_14 )
      Not()
      Coil( "DB1030_TEST_STOP".IS_PSP_ALARMS )
   END_RUNG
   RUNG wire#w1
      I_Contact( "DB1030_TEST_STOP".IS_PSP_ALARMS )
      I_Contact( "DB1030_TEST_STOP".TEST_STP_INTERNAL_P_F_AX_15 )
      I_Contact( "DB1030_TEST_STOP".TEST_STP_INTERNAL_P_F_AX_16 )
      I_Contact( "DB1030_TEST_STOP".TEST_STP_INTERNAL_P_F_AX_17 )
      I_Contact( "DB1030_TEST_STOP".TEST_STP_INTERNAL_P_F_AX_18 )
      I_Contact( "DB1030_TEST_STOP".TEST_STP_INTERNAL_P_F_AX_19 )
      I_Contact( "DB1030_TEST_STOP".TEST_STP_INTERNAL_P_F_AX_20 )
      I_Contact( "DB1030_TEST_STOP".TEST_STP_INTERNAL_P_F_AX_21 )
      Not()
      Coil( "DB1030_TEST_STOP".IS_PSP_ALARMS )
   END_RUNG
   RUNG wire#w1
      I_Contact( "DB1030_TEST_STOP".IS_PSP_ALARMS )
      I_Contact( "DB1030_TEST_STOP".TEST_STP_INTERNAL_P_F_AX_22 )
      I_Contact( "DB1030_TEST_STOP".TEST_STP_INTERNAL_P_F_AX_23 )
      I_Contact( "DB1030_TEST_STOP".TEST_STP_INTERNAL_P_F_AX_24 )
      I_Contact( "DB1030_TEST_STOP".TEST_STP_INTERNAL_P_F_AX_25 )
      I_Contact( "DB1030_TEST_STOP".TEST_STP_INTERNAL_P_F_AX_26 )
      I_Contact( "DB1030_TEST_STOP".TEST_STP_INTERNAL_P_F_AX_27 )
      I_Contact( "DB1030_TEST_STOP".TEST_STP_INTERNAL_P_F_AX_28 )
      Not()
      Coil( "DB1030_TEST_STOP".IS_PSP_ALARMS )
   END_RUNG
   RUNG wire#w1
      I_Contact( "DB1030_TEST_STOP".IS_PSP_ALARMS )
      I_Contact( "DB1030_TEST_STOP".TEST_STP_INTERNAL_P_F_AX_29 )
      I_Contact( "DB1030_TEST_STOP".TEST_STP_INTERNAL_P_F_AX_30 )
      I_Contact( "DB1030_TEST_STOP".TEST_STP_INTERNAL_P_F_AX_31 )
      Not()
      Coil( "DB1030_TEST_STOP".IS_PSP_ALARMS )
   END_RUNG
   // the same network as SCL:
   "DB1030_TEST_STOP".IS_PSP_ALARMS := NOT ("M_ONE" AND NOT "DB1030_TEST_STOP".TEST_STP_SQ_TIME_EXCEEDED AND NOT "DB1030_TEST_STOP".TEST_STP_TST_BRK_F_AX_1 AND NOT "DB1030_TEST_STOP".TEST_STP_TST_BRK_F_AX_2 AND NOT "DB1030_TEST_STOP".TEST_STP_TST_BRK_F_AX_3 AND NOT "DB1030_TEST_STOP".TEST_STP_TST_BRK_F_AX_4 AND NOT "DB1030_TEST_STOP".TEST_STP_TST_BRK_F_AX_5 AND NOT "DB1030_TEST_STOP".TEST_STP_TST_BRK_F_AX_6);
   "DB1030_TEST_STOP".IS_PSP_ALARMS := NOT ("M_ONE" AND NOT "DB1030_TEST_STOP".IS_PSP_ALARMS AND NOT "DB1030_TEST_STOP".TEST_STP_INTERNAL_P_F_AX_1 AND NOT "DB1030_TEST_STOP".TEST_STP_INTERNAL_P_F_AX_2 AND NOT "DB1030_TEST_STOP".TEST_STP_INTERNAL_P_F_AX_3 AND NOT "DB1030_TEST_STOP".TEST_STP_INTERNAL_P_F_AX_4 AND NOT "DB1030_TEST_STOP".TEST_STP_INTERNAL_P_F_AX_5 AND NOT "DB1030_TEST_STOP".TEST_STP_INTERNAL_P_F_AX_6 AND NOT "DB1030_TEST_STOP".TEST_STP_INTERNAL_P_F_AX_7);
   "DB1030_TEST_STOP".IS_PSP_ALARMS := NOT ("M_ONE" AND NOT "DB1030_TEST_STOP".IS_PSP_ALARMS AND NOT "DB1030_TEST_STOP".TEST_STP_INTERNAL_P_F_AX_8 AND NOT "DB1030_TEST_STOP".TEST_STP_INTERNAL_P_F_AX_9 AND NOT "DB1030_TEST_STOP".TEST_STP_INTERNAL_P_F_AX_10 AND NOT "DB1030_TEST_STOP".TEST_STP_INTERNAL_P_F_AX_11 AND NOT "DB1030_TEST_STOP".TEST_STP_INTERNAL_P_F_AX_12 AND NOT "DB1030_TEST_STOP".TEST_STP_INTERNAL_P_F_AX_13 AND NOT "DB1030_TEST_STOP".TEST_STP_INTERNAL_P_F_AX_14);
   "DB1030_TEST_STOP".IS_PSP_ALARMS := NOT ("M_ONE" AND NOT "DB1030_TEST_STOP".IS_PSP_ALARMS AND NOT "DB1030_TEST_STOP".TEST_STP_INTERNAL_P_F_AX_15 AND NOT "DB1030_TEST_STOP".TEST_STP_INTERNAL_P_F_AX_16 AND NOT "DB1030_TEST_STOP".TEST_STP_INTERNAL_P_F_AX_17 AND NOT "DB1030_TEST_STOP".TEST_STP_INTERNAL_P_F_AX_18 AND NOT "DB1030_TEST_STOP".TEST_STP_INTERNAL_P_F_AX_19 AND NOT "DB1030_TEST_STOP".TEST_STP_INTERNAL_P_F_AX_20 AND NOT "DB1030_TEST_STOP".TEST_STP_INTERNAL_P_F_AX_21);
   "DB1030_TEST_STOP".IS_PSP_ALARMS := NOT ("M_ONE" AND NOT "DB1030_TEST_STOP".IS_PSP_ALARMS AND NOT "DB1030_TEST_STOP".TEST_STP_INTERNAL_P_F_AX_22 AND NOT "DB1030_TEST_STOP".TEST_STP_INTERNAL_P_F_AX_23 AND NOT "DB1030_TEST_STOP".TEST_STP_INTERNAL_P_F_AX_24 AND NOT "DB1030_TEST_STOP".TEST_STP_INTERNAL_P_F_AX_25 AND NOT "DB1030_TEST_STOP".TEST_STP_INTERNAL_P_F_AX_26 AND NOT "DB1030_TEST_STOP".TEST_STP_INTERNAL_P_F_AX_27 AND NOT "DB1030_TEST_STOP".TEST_STP_INTERNAL_P_F_AX_28);
   "DB1030_TEST_STOP".IS_PSP_ALARMS := NOT ("M_ONE" AND NOT "DB1030_TEST_STOP".IS_PSP_ALARMS AND NOT "DB1030_TEST_STOP".TEST_STP_INTERNAL_P_F_AX_29 AND NOT "DB1030_TEST_STOP".TEST_STP_INTERNAL_P_F_AX_30 AND NOT "DB1030_TEST_STOP".TEST_STP_INTERNAL_P_F_AX_31);
END_REGION

REGION Network 99: IMMEDIATE STOP ALARMS
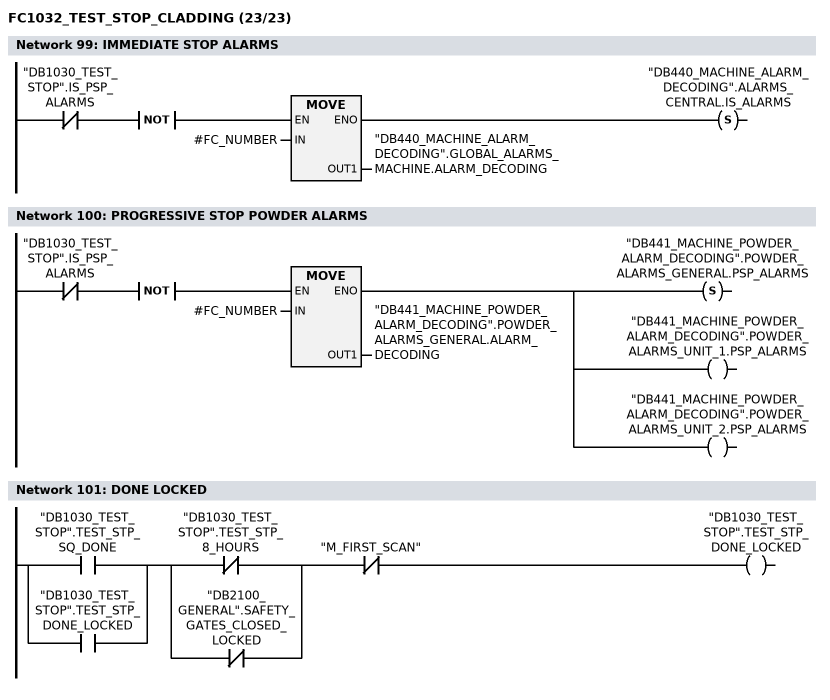
   RUNG wire#powerrail
      I_Contact( "DB1030_TEST_STOP".IS_PSP_ALARMS )
      Not()
      { S7_GenerateENO := "TRUE" } Move(in := #FC_NUMBER, out1 => "DB440_MACHINE_ALARM_DECODING".GLOBAL_ALARMS_MACHINE.ALARM_DECODING)
      S_Coil( "DB440_MACHINE_ALARM_DECODING".ALARMS_CENTRAL.IS_ALARMS )
   END_RUNG
   // the same network as SCL:
   // ENO of a box is taken as its EN; it also drops when the box reports an error
   IF NOT (NOT "DB1030_TEST_STOP".IS_PSP_ALARMS) THEN
       "DB440_MACHINE_ALARM_DECODING".GLOBAL_ALARMS_MACHINE.ALARM_DECODING := #FC_NUMBER;
       "DB440_MACHINE_ALARM_DECODING".ALARMS_CENTRAL.IS_ALARMS := TRUE;
   END_IF;
END_REGION

REGION Network 100: PROGRESSIVE STOP POWDER ALARMS
   RUNG wire#powerrail
      I_Contact( "DB1030_TEST_STOP".IS_PSP_ALARMS )
      Not()
      { S7_GenerateENO := "TRUE" } Move(in := #FC_NUMBER, out1 => "DB441_MACHINE_POWDER_ALARM_DECODING".POWDER_ALARMS_GENERAL.ALARM_DECODING)
      wire#w1
      S_Coil( "DB441_MACHINE_POWDER_ALARM_DECODING".POWDER_ALARMS_GENERAL.PSP_ALARMS )
   END_RUNG
   RUNG wire#w1
      Coil( "DB441_MACHINE_POWDER_ALARM_DECODING".POWDER_ALARMS_UNIT_1.PSP_ALARMS )
   END_RUNG
   RUNG wire#w1
      Coil( "DB441_MACHINE_POWDER_ALARM_DECODING".POWDER_ALARMS_UNIT_2.PSP_ALARMS )
   END_RUNG
   // the same network as SCL:
   // ENO of a box is taken as its EN; it also drops when the box reports an error
   #_w1 := NOT (NOT "DB1030_TEST_STOP".IS_PSP_ALARMS);
   IF #_w1 THEN
       "DB441_MACHINE_POWDER_ALARM_DECODING".POWDER_ALARMS_GENERAL.ALARM_DECODING := #FC_NUMBER;
       "DB441_MACHINE_POWDER_ALARM_DECODING".POWDER_ALARMS_GENERAL.PSP_ALARMS := TRUE;
   END_IF;
   "DB441_MACHINE_POWDER_ALARM_DECODING".POWDER_ALARMS_UNIT_1.PSP_ALARMS := #_w1;
   "DB441_MACHINE_POWDER_ALARM_DECODING".POWDER_ALARMS_UNIT_2.PSP_ALARMS := #_w1;
END_REGION

REGION Network 101: DONE LOCKED
   RUNG wire#powerrail
      Contact( "DB1030_TEST_STOP".TEST_STP_SQ_DONE )
      wire#w1
      I_Contact( "DB1030_TEST_STOP".TEST_STP_8_HOURS )
      wire#w2
      I_Contact( "M_FIRST_SCAN" )
      Coil( "DB1030_TEST_STOP".TEST_STP_DONE_LOCKED )
   END_RUNG
   RUNG wire#powerrail
      Contact( "DB1030_TEST_STOP".TEST_STP_DONE_LOCKED )
   END_RUNG wire#w1
   RUNG wire#w1
      I_Contact( "DB2100_GENERAL".SAFETY_GATES_CLOSED_LOCKED )
   END_RUNG wire#w2
   // the same network as SCL:
   "DB1030_TEST_STOP".TEST_STP_DONE_LOCKED := ("DB1030_TEST_STOP".TEST_STP_SQ_DONE OR "DB1030_TEST_STOP".TEST_STP_DONE_LOCKED) AND (NOT "DB1030_TEST_STOP".TEST_STP_8_HOURS OR NOT "DB2100_GENERAL".SAFETY_GATES_CLOSED_LOCKED) AND NOT "M_FIRST_SCAN";
END_REGION
END_FUNCTION
